# EPICS substitutions: bpm_data_combiner_app/Db/bpm_names_mls_gen.substitutions
file "db/bpm_names_mls_rec.db"
{
	pattern { SEC_TYP SEC_NUM }
		{ K       3       }
		{ L       4       }
		{ K       1       }
		{ L       2       }
}
